# EPICS autosave request: support/ip/2-9/ipApp/Db/SR630_settings.req
$(P)$(R)$(N).DESC
$(P)$(R)$(N)_READ.SCAN
